# B&R Automation Studio project PT_KB_V01 (part 6)

#### ProcessValues.st
```iecst
ACTION ProcessValues:
	(* ======================================================================== *)
	(* 1) Izbor realnog protoka aktivnog izvora                                 *)
	(* ======================================================================== *)
	CASE PGRad.Ctrl.SelektovaniIzvor OF
		_01_BRB2:
			AktivniUlazniProtok := PG01_Remote.BRB2Sens.FtRB21.Value;

		_02_IEBKB1:
			AktivniUlazniProtok := IEB_KB1.Cntrl.Comm.Podstanica.Status.TrenutniProtok;

	ELSE
		AktivniUlazniProtok := 0.0;
	END_CASE

	(* ======================================================================== *)
	(* 2) Toplotne snage                                                        *)
	(* ======================================================================== *)
	Predata_Snaga := 4.181 * AktivniUlazniProtok
		* (PG.Sens.Tt._1.AI_Output.ScaledValue - PG.Sens.Tt._2.AI_Output.ScaledValue);
	Snaga_grejanja_hotela := 4.181 * AktivniUlazniProtok
		* (PG.Sens.Tt._1.AI_Output.ScaledValue - PG.Sens.Tt._4.AI_Output.ScaledValue);
	Snaga_sanitarnog_grejanja := Predata_Snaga - Snaga_grejanja_hotela;

	(* ======================================================================== *)
	(* 3) Ostale izvedene procesne velicine                                     *)
	(* ======================================================================== *)
	NivoPRihvatniSud := (PG.Sens.Pt._NS1.AI_Output.ScaledValue - PG.Sens.Pt._NS2.AI_Output.ScaledValue) / 0.09804;
	DP_strainer := PG.Sens.Pt._1.AI_Output.ScaledValue - PG.Sens.Pt._2.AI_Output.ScaledValue + 0.123;
	DP_Izmejnivac := PG.Sens.Pt._2.AI_Output.ScaledValue - PG.Sens.Pt._3.AI_Output.ScaledValue + 0.0015;
END_ACTION
```

### Program Logical/PID_Pu_01 (IEC)

#### Variables.var
```iecst
VAR
	Start_Pu_01 : BOOL;
END_VAR
```

#### Cyclic.st
```iecst
PROGRAM _CYCLIC
	(* ======================================================================== *)
	(* PID_Pu_01_CYCLIC                                                          *)
	(* Zatvorena petlja nivoa: ActValue uzima nivo prihvatnog suda,              *)
	(* a izlaz PID-a se, kada je dozvoljeno startPIDPu1, mapira na Pu._1 freq.   *)
	(* ======================================================================== *)

	(* -------------------------------------------------------------------------- *)
	(* 1) Rad po komandi state masine: PID je jedini vlasnik frekvencije i Run-a. *)
	(* -------------------------------------------------------------------------- *)
	IF PGRad_Cmd.Aktivan THEN
		Start_Pu_01 := FALSE;
		startPIDPu1 := PGRad_Cmd.PID.Enable;

		(* 1.1) Prenos procesnog zahteva u PID regulator. *)
		PID_Pu_01.Enable := PGRad_Cmd.PID.Enable;
		PID_Pu_01.ActValue := PGRad_Cmd.PID.ActValue;
		PID_Pu_01.SetValue := PGRad_Cmd.PID.SetValue;
		PID_Pu_01.Invert := PGRad_Cmd.PID.Invert;
		PID_Pu_01.MaxOut := PGRad_Cmd.PID.MaxOut;
		PID_Pu_01.EnableTracking := PGRad_Cmd.PID.EnableTracking;
		PID_Pu_01.TrackingValue := PGRad_Cmd.PID.TrackingValue;
		IF EDGEPOS(PGRad_Cmd.PID.Enable) THEN
			PID_Pu_01.Update := TRUE;
		END_IF
		PID_Pu_01();
		IF PID_Pu_01.UpdateDone THEN
			PID_Pu_01.Update := FALSE;
		END_IF

		(* 1.2) Iskljucivo izabrana izlazna pumpa dobija PID frekvenciju i Run. *)
		PG.Act.Pu._1.cmds.Run_fwd := FALSE;
		PG.Act.Pu._2.cmds.Run_fwd := FALSE;
		IF PGRad_Cmd.PID.Enable THEN
			IF PGRad_Cmd.Pumpe._01.Run THEN
				PG.Act.Pu._1.params.Freq := PID_Pu_01.Out;
				PG.Act.Pu._1.cmds.Run_fwd := TRUE;
			ELSIF PGRad_Cmd.Pumpe._02.Run THEN
				PG.Act.Pu._2.params.Freq := PID_Pu_01.Out;
				PG.Act.Pu._2.cmds.Run_fwd := TRUE;
			END_IF
		END_IF

	ELSE
		(* -------------------------------------------------------------------------- *)
		(* 2) Nasledjeni rucni/auto rad pumpe 1                                    *)
		(* -------------------------------------------------------------------------- *)
		(* 2.1) Ciklicni PID poziv sa nivoom prihvatnog suda kao merenom vrednoscu. *)
		PID_Pu_01.EnableTracking := FALSE;
		PID_Pu_01.ActValue := NivoPRihvatniSud;
		PID_Pu_01();

		IF startPIDPu1 THEN
			PG.Act.Pu._1.params.Freq := PID_Pu_01.Out;
		END_IF

		(* 2.2) Automatski start/stop iz nivoa i rucne komande. *)
		IF Pu_01_Auto THEN
			IF NivoPRihvatniSud > PID_Pu_01.SetValue THEN
				Start_Pu_01 := TRUE;
				startPIDPu1 := TRUE;
				PG.Act.AV._3.Open := TRUE;
			ELSIF (NivoPRihvatniSud < (PID_Pu_01.SetValue - 0.6))
				OR (NivoPRihvatniSud < 0.75) THEN
				Start_Pu_01 := FALSE;
				startPIDPu1 := FALSE;
				PG.Act.AV._3.Open := FALSE;
			END_IF
		END_IF

		IF EDGENEG(Pu_01_Auto) THEN
			Start_Pu_01 := FALSE;
		END_IF

		IF EDGEPOS(Start_Pu_01) THEN
			PID_Pu_01.Update := TRUE;
		END_IF

		(* 2.3) Primena Run komande i reset PID dozvole na ivicama zahteva. *)
		IF Start_Pu_01 THEN
			PID_Pu_01.Enable := TRUE;
			PG.Act.Pu._1.cmds.Run_fwd := TRUE;

			IF PID_Pu_01.UpdateDone THEN
				PID_Pu_01.Update := FALSE;
			END_IF
		END_IF

		IF EDGENEG(Start_Pu_01) THEN
			PID_Pu_01.Enable := FALSE;
			PG.Act.Pu._1.cmds.Run_fwd := FALSE;
		END_IF

		(* -------------------------------------------------------------------------- *)
		(* 3) Zadrzavanje otvorenog izlaznog ventila                                *)
		(* -------------------------------------------------------------------------- *)
		(* PG_V05 prati otvoren ulazni ventil PG_V01 u nasledjenom lokalnom rezimu. *)
		IF PG.Act.AV._1.Open THEN
			PG.Act.AV._5.Open := TRUE;
		END_IF
	END_IF
END_PROGRAM
```

#### Exit.st
```iecst
PROGRAM _EXIT
	(* ======================================================================== *)
	(* PID_Pu_01_EXIT                                                            *)
	(* Nema posebne EXIT akcije; Run i frekvencu vlasnicki postavlja CYCLIC.     *)
	(* ======================================================================== *)

END_PROGRAM
```

#### Init.st
```iecst
PROGRAM _INIT
	(* ======================================================================== *)
	(* PID_Pu_01_INIT                                                            *)
	(* U ovom tasku trenutno nema inicijalizacionih dodela.                      *)
	(* Retain procesni parametri se postavljaju iz HMI/visih nivoa logike.       *)
	(* ======================================================================== *)
	(* -------------------------------------------------------------------------- *)
	(* 1) Inicijalni parametri PID izlazne pumpe                                  *)
	(* -------------------------------------------------------------------------- *)
	(* Frekvencija izlazne pumpe je ogranicena na radni opseg 20.0..70.0 Hz. *)
	PID_Pu_01.MaxOut := 70.0; (* Gornja granica PID izlaza [Hz]. *)
	PID_Pu_01.MinOut := 20.0; (* Donja granica PID izlaza [Hz]. *)

	(* Parametri nivo regulacije; D deo je iskljucen, a filter prigusuje merenje. *)
	PID_Pu_01.PIDParameters.DerivativeTime := 0.0; (* D vreme [s]. *)
	PID_Pu_01.PIDParameters.FilterTime := 45.0; (* Filter merenja [s]. *)
	PID_Pu_01.PIDParameters.Gain := 96.3; (* Proporcionalno pojacanje. *)
	PID_Pu_01.PIDParameters.IntegrationTime := 180; (* Integraciono vreme [s]. *)
	PID_Pu_01.Invert := TRUE; (* Nivo regulacija koristi inverzni smer. *)

	PID_Pu_01.SetValue := 1.5; (* Lokalni pocetni setpoint nivoa [m]. *)

END_PROGRAM
```

### Program Logical/Rad_PG_KB (IEC)

#### Variables.var
```iecst
VAR
	(* Izvrsni kontekst state masine. *)
	State : E_PGRad_State := PG_00_Stand_By; (* Trenutni korak state masine *)
	Substep : USINT := 0; (* Podkorak aktivnog stanja: 0 = ulazak, 1..N = izvrsavanje *)

	(* HMI komande. *)
	KomandaStart : BOOL; (* HMI komanda za pokretanje sistema *)
	KomandaStop : BOOL; (* HMI komanda za kontrolisano zaustavljanje *)
	KomandaReset : BOOL; (* HMI komanda za reset uklonjene greske *)
	SelectIEBKB1 : BOOL; (* HMI Toggle: FALSE = BRB2, TRUE = IEBKB1; prihvata se samo u Standby. *)
	ManualMode : BOOL; (* Servisni rucni rezim; dozvoljen samo iz Standby. *)
	ManualSequence : USINT; (* Izabrana sekvenca servisnog rada. *)
	ManualStart : BOOL; (* Impuls za pokretanje izabrane sekvence. *)
	ManualStop : BOOL; (* Impuls za kontrolisani prekid servisne sekvence. *)
	ManualNextStep : BOOL; (* Impuls za sledeci dozvoljeni podkorak. *)
	ManualAbort : BOOL; (* Impuls za povratak u Standby. *)
	CmdSetDefaultParameters : BOOL; (* Jednokratno vracanje svih parametara na projektne default vrednosti *)

	(* Dijagnostika aktivne greske. *)
	FaultLatched : BOOL; (* Aktivna zakacena greska, zahteva reset nakon otklanjanja uzroka *)
	FaultCode : USINT; (* Sifra aktivne greske za HMI i AsIMA *)
	FaultText : STRING[80]; (* Tekst aktivne greske za HMI *)

	(* Nadzor polozaja ventila i protoka izvora. *)
	T_PG_V01_Close : TON; (* Timeout zatvaranja IEBKB1 dovodnog ventila. *)
	T_PG_V01_Open : TON; (* Timeout otvaranja IEBKB1 dovodnog ventila. *)
	T_PG_V02_Open : TON; (* Timeout otvaranja BRB2 dovodnog ventila pri pripremi BRB2. *)
	T_PG_V02_Close : TON; (* Timeout zatvaranja BRB2 dovodnog ventila pri pripremi IEBKB1. *)
	T_IEBKB1_StartProtokTimeout : TON; (* Maksimalno cekanje pocetka IEBKB1 dotoka nakon otvaranja PG_V05. *)
	T_IEBKB1_ProtokNula : TON; (* Debounce potvrda protoka manjeg od 0.1 l/s. *)
	T_IEBKB1_StopProtokTimeout : TON; (* Maksimalno cekanje prestanka IEBKB1 dotoka pre zatvaranja PG_V05. *)
	T_PG_V05_Close : TON; (* Timeout zatvaranja PG_V05 nakon potvrdenog prestanka IEBKB1 dotoka. *)

	(* PID regulatori i izvrsne pomocne vrednosti. *)
	T_PrelazPV05Cuvar : TON; (* Vreme mekane promene PT06 SP-a od preispiranja do cuvara instalacije. *)
	PID_PV05 : MTBasicsPID; (* PID PG_PV05: PT06 pritisak preispiranja i cuvara instalacije. *)
	PID_PV_UlazTanka : MTBasicsPID; (* PID aktivnog PG_PV01/PG_PV02: PT04 pritisak pri punjenju tanka. *)
	SP_PV05 : REAL; (* Trenutni rampirani PT06 SP za PID PG_PV05 [bar]. *)
	PV05IspiranjeOtvoreno : BOOL; (* PT06 je dostigao SP i PG_PV05 je dozvoljen za ispiranje. *)
	IzlaznaPumpaUStopu : BOOL; (* Pumpa nastavlja praznjenje tanka do donje granice hysteresis. *)
END_VAR
```

#### Cyclic.sfc
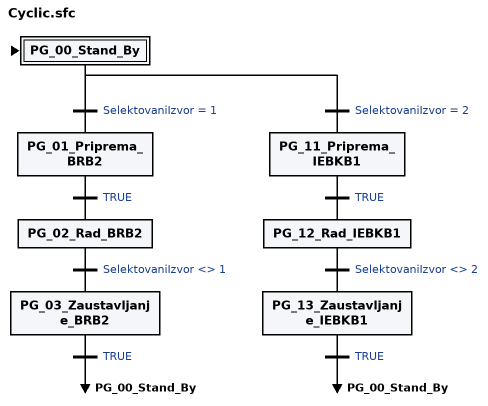
```iecst
PROGRAM _CYCLIC
INITIAL_STEP PG_00_Stand_By:
END_STEP
TRANSITION FROM PG_00_Stand_By TO PG_01_Priprema_BRB2:=
SelektovaniIzvor = 1
END_TRANSITION
TRANSITION FROM PG_00_Stand_By TO PG_11_Priprema_IEBKB1:=
SelektovaniIzvor = 2
END_TRANSITION
STEP PG_11_Priprema_IEBKB1:
END_STEP
TRANSITION FROM PG_11_Priprema_IEBKB1 TO PG_12_Rad_IEBKB1:=
TRUE
END_TRANSITION
STEP PG_12_Rad_IEBKB1:
END_STEP
TRANSITION FROM PG_12_Rad_IEBKB1 TO PG_13_Zaustavljanje_IEBKB1:=
SelektovaniIzvor <> 2
END_TRANSITION
STEP PG_13_Zaustavljanje_IEBKB1:
END_STEP
TRANSITION FROM PG_13_Zaustavljanje_IEBKB1 TO PG_00_Stand_By:=
TRUE
END_TRANSITION
(* @SFCISJUMP := 'PG_00_Stand_By' *)
STEP PG_01_Priprema_BRB2:
END_STEP
TRANSITION FROM PG_01_Priprema_BRB2 TO PG_02_Rad_BRB2:=
TRUE
END_TRANSITION
STEP PG_02_Rad_BRB2:
END_STEP
TRANSITION FROM PG_02_Rad_BRB2 TO PG_03_Zaustavljanje_BRB2:=
SelektovaniIzvor <> 1
END_TRANSITION
STEP PG_03_Zaustavljanje_BRB2:
END_STEP
TRANSITION FROM PG_03_Zaustavljanje_BRB2 TO PG_00_Stand_By:=
TRUE
END_TRANSITION
(* @SFCISJUMP := 'PG_00_Stand_By' *)
END_PROGRAM
```

#### Cyclic.st
```iecst
PROGRAM _CYCLIC
	(* ======================================================================== *)
	(* Rad_PG_KB_CYCLIC                                                          *)
	(* State masina izbora i rada izvora termalne vode: BRB2 (1) ili IEBKB1 (2). *)
	(* Prelazak izmedju grana ide iskljucivo preko PG_00_Stand_By - direktan     *)
	(* prelazak 1->2 ili 2->1 nije moguc.                                       *)
	(* ======================================================================== *)

	(* -------------------------------------------------------------------------- *)
	(* 1) Vracanje projektnih podrazumevanih parametara                          *)
	(* -------------------------------------------------------------------------- *)
	IF CmdSetDefaultParameters THEN
		PGRad.Par.SetPritisakPotisa := 1.5;
		PGRad.Par.MinProtok := 2.0;
		PGRad.Par.MaxProtok := 16.2;
		PGRad.Par.MinFR_Pumpe := 2.0;
		PGRad.Par.MaxFR_Pumpe := 16.2;
		PGRad.Par.SetPointNivoTanka := 1.5;
		PGRad.Par.SetPointMinTempIspiranja := 60.0;
		PGRad.Par.SetPointPritisakPV05Ispiranje := 5.5;
		PGRad.Par.SetPointPritisakUlazTanka := 5.5;
		PGRad.Par.SetPointMaxPritisakDolaznaCev := 6.5;
		PGRad.Par.TimeSP.PrelazPV05Cuvar_s := 15.0;
		PGRad.Par.PocetnaFrekvencaIzlaznePumpe := 20.0;
		PGRad.Par.MaxOtvorPropZaZatvaranje := 0.1;
		PGRad.Par.TimeSP.OverlapPumpi_s := 10.0;
		PGRad.Par.TimeSP.AutoRestartDelay_s := 60.0;
		PGRad.Par.TimeSP.ValvePositionTimeout_s := 30.0;
		PGRad.Par.TimeSP.InterlockDebounce_s := 2.0;

		(* BRB2 odzracivanje: oba ventila, prag 1.5 bar sa 0.5 bar histerezom. *)
		PGRad.Par.AirRelease.BRB2.PV03.NumberOfLS := 2;
		PGRad.Par.AirRelease.BRB2.PV03.PressureSP_bar := 1.5;
		PGRad.Par.AirRelease.BRB2.PV03.PressureHysteresis_bar := 0.5;
		PGRad.Par.AirRelease.BRB2.PV03.LS1.SP_Percent := 20.0;
		PGRad.Par.AirRelease.BRB2.PV03.LS1.Ramp_PercentPerSecond := 2.0;
		PGRad.Par.AirRelease.BRB2.PV03.LS1.ConfirmTime_s := 1.0;
		PGRad.Par.AirRelease.BRB2.PV03.LS2.SP_Percent := 89.0;
		PGRad.Par.AirRelease.BRB2.PV03.LS2.Ramp_PercentPerSecond := 15.0;
		PGRad.Par.AirRelease.BRB2.PV03.LS2.ConfirmTime_s := 1.0;
		PGRad.Par.AirRelease.BRB2.PV04 := PGRad.Par.AirRelease.BRB2.PV03;

		(* IEBKB1 odzracivanje: aktivan je PV03 sa nizim pragom pritiska. *)
		PGRad.Par.AirRelease.IEBKB1.PV03.NumberOfLS := 2;
		PGRad.Par.AirRelease.IEBKB1.PV03.PressureSP_bar := 0.15;
		PGRad.Par.AirRelease.IEBKB1.PV03.PressureHysteresis_bar := 0.05;
		PGRad.Par.AirRelease.IEBKB1.PV03.LS1.SP_Percent := 20.0;
		PGRad.Par.AirRelease.IEBKB1.PV03.LS1.Ramp_PercentPerSecond := 2.0;
		PGRad.Par.AirRelease.IEBKB1.PV03.LS1.ConfirmTime_s := 1.0;
		PGRad.Par.AirRelease.IEBKB1.PV03.LS2.SP_Percent := 89.0;
		PGRad.Par.AirRelease.IEBKB1.PV03.LS2.Ramp_PercentPerSecond := 15.0;
		PGRad.Par.AirRelease.IEBKB1.PV03.LS2.ConfirmTime_s := 1.0;
		PGRad.Par.AirRelease.IEBKB1.PV04 := PGRad.Par.AirRelease.IEBKB1.PV03;

		CmdSetDefaultParameters := FALSE;
	END_IF

	(* -------------------------------------------------------------------------- *)
	(* 2) Podrazumevane neretentivne komande po scan-u                            *)
	(* -------------------------------------------------------------------------- *)
	PGRad_Cmd.Aktivan := FALSE;
	PGRad_Cmd.Ventili._03_Open := FALSE;
	PGRad_Cmd.Ventili._04_Open := FALSE;
	PGRad_Cmd.Ventili._05_Open := FALSE;
	PGRad_Cmd.Ventili._06_Open := FALSE;
	PGRad_Cmd.Ventili._07_Open := FALSE;

	PGRad_Cmd.PropVentili.PV01.Enable := FALSE;
	PGRad_Cmd.PropVentili.PV01.SP_Percent := 0.0;
	PGRad_Cmd.PropVentili.PV02.Enable := FALSE;
	PGRad_Cmd.PropVentili.PV02.SP_Percent := 0.0;
	PGRad_Cmd.PropVentili.PV05.Enable := FALSE;
	PGRad_Cmd.PropVentili.PV05.SP_Percent := 0.0;
	PGRad_Cmd.AirRelease.PV03.Enable := FALSE;
	PGRad_Cmd.AirRelease.PV04.Enable := FALSE;
	PGRad_Cmd.AirRelease.UseIEBKB1Parameters := FALSE;
	PGRad_Cmd.AirRelease.ResetAll := KomandaReset;

	PGRad_Cmd.Pumpe._01.Run := FALSE;
	PGRad_Cmd.Pumpe._02.Run := FALSE;
	PGRad_Cmd.PID.Enable := FALSE;
	PGRad_Cmd.PID.ActValue := 0.0;
	PGRad_Cmd.PID.SetValue := 0.0;
	PGRad_Cmd.PID.Invert := FALSE;
	PGRad_Cmd.PID.MaxOut := 0.0;
	PGRad_Cmd.PID.EnableTracking := FALSE;
	PGRad_Cmd.PID.TrackingValue := 0.0;
	PGRad_BRB2Cmd.RadKaPodstanici := FALSE;
	PGRad_BRB2Cmd.ZahtevStarta := FALSE;
	PGRad_BRB2Cmd.ZahtevZaustavljanja := FALSE;
	PGRad_BRB2Cmd.ManualMode := ManualMode;
	PGRad_BRB2Cmd.ManualSequence := ManualSequence;
	PGRad_BRB2Cmd.ManualStart := ManualStart;
	PGRad_BRB2Cmd.ManualStop := ManualStop;
	PGRad_BRB2Cmd.ManualNextStep := ManualNextStep;
	PGRad_BRB2Cmd.ManualAbort := ManualAbort;
	PGRad_BRB2Cmd.VentiliPodstaniceZatvoreni := FALSE;
	PGRad_BRB2Cmd.PritisakIEBKB1 := IEB_KB1.Sens.Pt.B_02._01_value;
	PGRad_BRB2Cmd.PodstanicaURezimuRada := FALSE;
	IEB_KB1.Cntrl.Comm.Podstanica.Zahtev.ZahtevVode := FALSE;
	IEB_KB1.Cntrl.Comm.Podstanica.Zahtev.NivoPrihvatnogTanka := NivoPRihvatniSud;
	IEB_KB1.Cntrl.Comm.Podstanica.Zahtev.CiljaniProtok := PGRad.Par.MaxProtok;
	IEB_KB1.Cntrl.Comm.Podstanica.Zahtev.ModRada := 0;
	IEB_KB1.Cntrl.proba := FALSE;

	(* Izbor izvora sa HMI prihvata se samo u bezbednom Standby stanju. *)
	IF State = PG_00_Stand_By THEN
		IF SelectIEBKB1 THEN
			PGRad.Ctrl.SelektovaniIzvor := _02_IEBKB1;
		ELSE
			PGRad.Ctrl.SelektovaniIzvor := _01_BRB2;
		END_IF;
	ELSE
		SelectIEBKB1 := PGRad.Ctrl.SelektovaniIzvor = _02_IEBKB1;
	END_IF;

	(* -------------------------------------------------------------------------- *)
	(* 3) Tajmeri pripreme BRB2 dovodne putanje                                  *)
	(* -------------------------------------------------------------------------- *)
	T_PG_V01_Close.IN := FALSE;
	T_PG_V01_Close.PT := REAL_TO_TIME(PGRad.Par.TimeSP.ValvePositionTimeout_s * 1000.0);
	T_PG_V02_Open.IN := FALSE;
	T_PG_V02_Open.PT := REAL_TO_TIME(PGRad.Par.TimeSP.ValvePositionTimeout_s * 1000.0);
	T_PG_V02_Close.IN := FALSE;
	T_PG_V02_Close.PT := REAL_TO_TIME(PGRad.Par.TimeSP.ValvePositionTimeout_s * 1000.0);
	T_PG_V01_Open.IN := FALSE;
	T_PG_V01_Open.PT := REAL_TO_TIME(PGRad.Par.TimeSP.ValvePositionTimeout_s * 1000.0);
	T_IEBKB1_StartProtokTimeout.IN := FALSE;
	T_IEBKB1_StartProtokTimeout.PT := REAL_TO_TIME(PGRad.Par.TimeSP.ValvePositionTimeout_s * 1000.0);
	T_IEBKB1_ProtokNula.IN := FALSE;
	T_IEBKB1_ProtokNula.PT := REAL_TO_TIME(PGRad.Par.TimeSP.InterlockDebounce_s * 1000.0);
	T_IEBKB1_StopProtokTimeout.IN := FALSE;
	T_IEBKB1_StopProtokTimeout.PT := REAL_TO_TIME(PGRad.Par.TimeSP.ValvePositionTimeout_s * 1000.0);
	T_PG_V05_Close.IN := FALSE;
	T_PG_V05_Close.PT := REAL_TO_TIME(PGRad.Par.TimeSP.ValvePositionTimeout_s * 1000.0);
	T_PrelazPV05Cuvar.IN := FALSE;
	T_PrelazPV05Cuvar.PT := REAL_TO_TIME(PGRad.Par.TimeSP.PrelazPV05Cuvar_s * 1000.0);

	CASE State OF

		PG_00_Stand_By:
			(* Neretentivni vektor je bezbedno resetovan u sekciji 2; V01/V02 se ne menjaju. *)
			PV05IspiranjeOtvoreno := FALSE;
			(* Start je dozvoljen samo sa izabranim izvorom i regulacionom varijantom. *)
			IF ManualMode AND ManualStart AND (ManualSequence = 1) THEN
				PGRad.Ctrl.SelektovaniIzvor := _01_BRB2;
				ManualStart := FALSE;
				State := PG_01_Priprema_BRB2;
				Substep := 0;
			ELSIF ManualMode AND ManualStart AND (ManualSequence = 2) THEN
				PGRad.Ctrl.SelektovaniIzvor := _02_IEBKB1;
				ManualStart := FALSE;
				State := PG_11_Priprema_IEBKB1;
				Substep := 0;
			ELSIF KomandaStart
				AND (NOT ManualMode)
				AND (NOT FaultLatched)
				AND (PGRad.Ctrl.RegulacionaVarijanta <> _00_neaktivan)
				AND (PGRad.Ctrl.SelektovaniIzvor = _01_BRB2) THEN
				State := PG_01_Priprema_BRB2;
				Substep := 0;
			ELSIF KomandaStart
				AND (NOT FaultLatched)
				AND (PGRad.Ctrl.RegulacionaVarijanta <> _00_neaktivan)
				AND (PGRad.Ctrl.SelektovaniIzvor = _02_IEBKB1) THEN
				State := PG_11_Priprema_IEBKB1;
				Substep := 0;
			END_IF

		PG_01_Priprema_BRB2:
			IF ManualStop OR ManualAbort THEN
				KomandaStop := TRUE;
				ManualStop := FALSE;
				ManualAbort := FALSE;
			END_IF;
			PGRad_BRB2Cmd.RadKaPodstanici := TRUE;
			PGRad_BRB2Cmd.ZahtevStarta := TRUE;
			CASE Substep OF
				0:
					(* Prioritet BRB2: najpre zatvori dovod sa IEBKB1. *)
					PGRad.CmdRetain.V01_Open := FALSE;
					Substep := 1;

				1:
					(* Otvaranje BRB2 dovoda je dozvoljeno tek po potvrdi zatvorenog V01. *)
					PGRad.CmdRetain.V01_Open := FALSE;
					T_PG_V01_Close.IN := NOT PG.Act.AV._1.Closed;
					IF PG.Act.AV._1.Closed AND (NOT ManualMode OR ManualNextStep) THEN
						ManualNextStep := FALSE;
						PGRad.CmdRetain.V02_Open := TRUE;
						Substep := 2;
					ELSIF T_PG_V01_Close.Q THEN
						PGRad.CmdRetain.V01_Open := FALSE;
						PGRad.CmdRetain.V02_Open := FALSE;
						FaultLatched := TRUE;
						FaultCode := 11;
						FaultText := 'PG_V01 nije zatvoren za zadato vreme';
						State := PG_00_Stand_By;
						Substep := 0;
					END_IF

				2:
					(* Ceka se fizicka potvrda otvorenog BRB2 dovoda. *)
					PGRad.CmdRetain.V01_Open := FALSE;
					PGRad.CmdRetain.V02_Open := TRUE;
					T_PG_V02_Open.IN := NOT PG.Act.AV._2.Opened;
					IF PG.Act.AV._2.Opened AND (NOT ManualMode OR ManualNextStep) THEN
						ManualNextStep := FALSE;
						Substep := 3;
					ELSIF T_PG_V02_Open.Q THEN
						PGRad.CmdRetain.V01_Open := FALSE;
						PGRad.CmdRetain.V02_Open := FALSE;
						FaultLatched := TRUE;
						FaultCode := 12;
						FaultText := 'PG_V02 nije otvoren za zadato vreme';
						State := PG_00_Stand_By;
						Substep := 0;
					END_IF

				3:
					(* PG_PV05 se otvara nakon dostignutog PT06 pritiska; temperatura se proverava tek posle BRB2 minimuma. *)
					IF PG.Sens.Pt._6.AI_Output.ScaledValue >= PGRad.Par.SetPointPritisakPV05Ispiranje THEN
						PV05IspiranjeOtvoreno := TRUE;
					END_IF;
					IF PV05IspiranjeOtvoreno THEN
						PGRad_Cmd.Aktivan := TRUE;
						PGRad_Cmd.PropVentili.PV05.Enable := TRUE;
					END_IF;
					IF PGRad_BRB2.IspiranjeMinTrajanjeDostignuto
						AND (PG.Sens.Tt._7.AI_Output.ScaledValue >= PGRad.Par.SetPointMinTempIspiranja) THEN
						IF ManualMode AND NOT ManualNextStep THEN
							(* Manual mode holds the completed rinse step until operator confirmation. *)
						ELSE
							ManualNextStep := FALSE;
							IF ManualMode AND (ManualSequence = 1) THEN
								(* Manual flush ends here; controlled stop closes the BRB2 path. *)
								KomandaStop := TRUE;
								State := PG_03_Zaustavljanje_BRB2;
								Substep := 0;
							ELSE
								Substep := 4;
							END_IF
						END_IF
					END_IF

				4:
					(* Priprema puta ka tanku: otvara se samo ON/OFF ventil izabranog ulaznog PV-a. *)
					PGRad_Cmd.Aktivan := TRUE;
					PGRad_Cmd.PropVentili.PV05.Enable := TRUE;
					CASE PGRad.Ctrl.AktivniPropVentilUlazTanka OF
						_01_PG_PV01:
							PGRad_Cmd.Ventili._06_Open := TRUE;
							PGRad_Cmd.PropVentili.PV01.Enable := TRUE;
							Substep := 5;
						_02_PG_PV02:
							PGRad_Cmd.Ventili._07_Open := TRUE;
							PGRad_Cmd.PropVentili.PV02.Enable := TRUE;
							Substep := 5;
					END_CASE

				5:
					(* Mek prelaz: ulazni PV vodi PT04, a PT06 SP PG_PV05 raste 5.5 -> 6.5 bar. *)
					PGRad_Cmd.Aktivan := TRUE;
					PGRad_Cmd.PropVentili.PV05.Enable := TRUE;
					T_PrelazPV05Cuvar.IN := TRUE;
					CASE PGRad.Ctrl.AktivniPropVentilUlazTanka OF
						_01_PG_PV01:
							PGRad_Cmd.Ventili._06_Open := TRUE;
							PGRad_Cmd.PropVentili.PV01.Enable := TRUE;
						_02_PG_PV02:
							PGRad_Cmd.Ventili._07_Open := TRUE;
							PGRad_Cmd.PropVentili.PV02.Enable := TRUE;
					END_CASE
					IF T_PrelazPV05Cuvar.Q AND (NOT ManualMode OR ManualNextStep) THEN
						ManualNextStep := FALSE;
						Substep := 6;
					END_IF

				6:
					(* Punjenje tanka: PV05 je cuvar PT06, a aktivni ulazni PV odrzava PT04. *)
					PGRad_Cmd.Aktivan := TRUE;
					PGRad_Cmd.PropVentili.PV05.Enable := TRUE;
					CASE PGRad.Ctrl.AktivniPropVentilUlazTanka OF
						_01_PG_PV01:
							PGRad_Cmd.Ventili._06_Open := TRUE;
							PGRad_Cmd.PropVentili.PV01.Enable := TRUE;
						_02_PG_PV02:
							PGRad_Cmd.Ventili._07_Open := TRUE;
							PGRad_Cmd.PropVentili.PV02.Enable := TRUE;
					END_CASE
					IF (NivoPRihvatniSud >= PGRad.Par.SetPointNivoTanka)
						AND (NOT ManualMode OR ManualNextStep) THEN
						ManualNextStep := FALSE;
						State := PG_02_Rad_BRB2;
						Substep := 0;
					END_IF

			ELSE
				Substep := 0;
			END_CASE

		PG_02_Rad_BRB2:
			PGRad_BRB2Cmd.RadKaPodstanici := TRUE;
			PGRad_BRB2Cmd.ZahtevStarta := TRUE;
			(* Odrzava PID regulaciju ulaza i PT06 cuvara nakon punjenja tanka. *)
			PGRad_Cmd.Aktivan := TRUE;
			PGRad_Cmd.PropVentili.PV05.Enable := TRUE;
			CASE PGRad.Ctrl.AktivniPropVentilUlazTanka OF
				_01_PG_PV01:
					PGRad_Cmd.Ventili._06_Open := TRUE;
					PGRad_Cmd.PropVentili.PV01.Enable := TRUE;
				_02_PG_PV02:
					PGRad_Cmd.Ventili._07_Open := TRUE;
					PGRad_Cmd.PropVentili.PV02.Enable := TRUE;
			END_CASE

			(* Izlaznu pumpu pokrece i frekvencu vodi iskljucivo PID_Pu_01. *)
			CASE PGRad.Ctrl.RegulacionaVarijanta OF
				_01_REG_PRITISAK:
					PGRad_Cmd.PID.Enable := TRUE;
					PGRad_Cmd.PID.ActValue := PG.Sens.Pt._5.AI_Output.ScaledValue;
					PGRad_Cmd.PID.SetValue := PGRad.Par.SetPritisakPotisa;
					PGRad_Cmd.PID.Invert := FALSE;
				_02_REG_NIVO:
					PGRad_Cmd.PID.Enable := TRUE;
					PGRad_Cmd.PID.ActValue := NivoPRihvatniSud;
					PGRad_Cmd.PID.SetValue := PGRad.Par.SetPointNivoTanka;
					PGRad_Cmd.PID.Invert := TRUE;
			END_CASE

			IF PGRad_Cmd.PID.Enable THEN
				PGRad_Cmd.PID.TrackingValue := PGRad.Par.PocetnaFrekvencaIzlaznePumpe;
				PGRad_Cmd.PID.EnableTracking := (Substep = 0);
				CASE PGRad.Ctrl.AktivnaPumpaIzlazTanka OF
					_01_Pu_PG_01:
						PGRad_Cmd.Ventili._03_Open := TRUE;
						PGRad_Cmd.Pumpe._01.Run := TRUE;
						PGRad_Cmd.PID.MaxOut := 70.0;
					_02_Pu_PG_02:
						PGRad_Cmd.Ventili._04_Open := TRUE;
						PGRad_Cmd.Pumpe._02.Run := TRUE;
						PGRad_Cmd.PID.MaxOut := 50.0;
				END_CASE
				Substep := 1;
			END_IF

			(* BRB2 sme preci u rad tek kada je tank pun i izabrana PG pumpa stvarno radi. *)
			PGRad_BRB2Cmd.PodstanicaURezimuRada :=
				(NivoPRihvatniSud >= PGRad.Par.SetPointNivoTanka)
				AND (
					((PGRad.Ctrl.AktivnaPumpaIzlazTanka = _01_Pu_PG_01)
						AND PG.Act.Pu._1.states.RUN)
					OR ((PGRad.Ctrl.AktivnaPumpaIzlazTanka = _02_Pu_PG_02)
						AND PG.Act.Pu._2.states.RUN)
				);

			(* Napusta granu cim PGRad.Ctrl.SelektovaniIzvor vise nije _01_BRB2. *)
			IF KomandaStop OR (PGRad.Ctrl.SelektovaniIzvor <> _01_BRB2) THEN
				State := PG_03_Zaustavljanje_BRB2;
				Substep := 0;
			END_IF

		PG_03_Zaustavljanje_BRB2:
			(* PT najpre trazi BRB2 ramp-down, zatim zatvara PV grane po stop SP potvrdi. *)
			PGRad_Cmd.Aktivan := TRUE;
			PGRad_BRB2Cmd.ZahtevZaustavljanja := TRUE;

			IF Substep = 0 THEN
				IzlaznaPumpaUStopu := TRUE;
				Substep := 1;
			END_IF;

			(* Izlazna pumpa ostaje na aktivnoj regulaciji dok tank ne padne ispod 60% SP-a. *)
			IF NivoPRihvatniSud < (0.6 * PGRad.Par.SetPointNivoTanka) THEN
				IzlaznaPumpaUStopu := FALSE;
			END_IF;

			IF IzlaznaPumpaUStopu THEN
				CASE PGRad.Ctrl.RegulacionaVarijanta OF
					_01_REG_PRITISAK:
						PGRad_Cmd.PID.Enable := TRUE;
						PGRad_Cmd.PID.ActValue := PG.Sens.Pt._5.AI_Output.ScaledValue;
						PGRad_Cmd.PID.SetValue := PGRad.Par.SetPritisakPotisa;
						PGRad_Cmd.PID.Invert := FALSE;
					_02_REG_NIVO:
						PGRad_Cmd.PID.Enable := TRUE;
						PGRad_Cmd.PID.ActValue := NivoPRihvatniSud;
						PGRad_Cmd.PID.SetValue := PGRad.Par.SetPointNivoTanka;
						PGRad_Cmd.PID.Invert := TRUE;
				END_CASE

				CASE PGRad.Ctrl.AktivnaPumpaIzlazTanka OF
					_01_Pu_PG_01:
						PGRad_Cmd.Ventili._03_Open := TRUE;
						PGRad_Cmd.Pumpe._01.Run := TRUE;
						PGRad_Cmd.PID.MaxOut := 70.0;
					_02_Pu_PG_02:
						PGRad_Cmd.Ventili._04_Open := TRUE;
						PGRad_Cmd.Pumpe._02.Run := TRUE;
						PGRad_Cmd.PID.MaxOut := 50.0;
				END_CASE
			END_IF;

			IF NOT PGRad_BRB2.StopSPDostignut THEN
				(* Dok BRB2 spusta frekvenciju, PT06 i PT04 ostaju u regulaciji. *)
				PGRad_Cmd.PropVentili.PV05.Enable := TRUE;
				CASE PGRad.Ctrl.AktivniPropVentilUlazTanka OF
					_01_PG_PV01:
						PGRad_Cmd.Ventili._06_Open := TRUE;
						PGRad_Cmd.PropVentili.PV01.Enable := TRUE;
					_02_PG_PV02:
						PGRad_Cmd.Ventili._07_Open := TRUE;
						PGRad_Cmd.PropVentili.PV02.Enable := TRUE;
				END_CASE
			END_IF;

			(* Nakon BRB2 stop SP-a svi proporcionalni ventili ostaju bez zahteva. *)
			PGRad_BRB2Cmd.VentiliPodstaniceZatvoreni := PGRad_BRB2.StopSPDostignut
				AND (PG.Act.PV._1.PV_Output.PV_Percent <= PGRad.Par.MaxOtvorPropZaZatvaranje)
				AND (PG.Act.PV._2.PV_Output.PV_Percent <= PGRad.Par.MaxOtvorPropZaZatvaranje)
				AND (PG.Act.PV._5.PV_Output.PV_Percent <= PGRad.Par.MaxOtvorPropZaZatvaranje);

			IF PGRad_BRB2.RB2V02Zatvoren AND NOT IzlaznaPumpaUStopu THEN
				State := PG_00_Stand_By;
				Substep := 0;
			END_IF

		PG_11_Priprema_IEBKB1:
			(* IEBKB1 put koristi samo PG_V01 i PG_V05; PV01/PV02/V06/V07 ostaju zatvoreni. *)
			IEB_KB1.Cntrl.Comm.Podstanica.Zahtev.ZahtevVode := TRUE;
			IEB_KB1.Cntrl.Comm.Podstanica.Zahtev.ModRada := 1;
			IEB_KB1.Cntrl.proba := TRUE;
			CASE Substep OF
				0:
					PGRad.CmdRetain.V02_Open := FALSE;
					Substep := 1;

				1:
					PGRad.CmdRetain.V02_Open := FALSE;
					T_PG_V02_Close.IN := NOT PG.Act.AV._2.Closed;
					IF PG.Act.AV._2.Closed THEN
						PGRad.CmdRetain.V01_Open := TRUE;
						Substep := 2;
					ELSIF T_PG_V02_Close.Q THEN
						PGRad.CmdRetain.V01_Open := FALSE;
						PGRad.CmdRetain.V02_Open := FALSE;
						FaultLatched := TRUE;
						FaultCode := 13;
						FaultText := 'PG_V02 nije zatvoren za zadato vreme';
						State := PG_00_Stand_By;
						Substep := 0;
					END_IF

				2:
					PGRad.CmdRetain.V01_Open := TRUE;
					PGRad.CmdRetain.V02_Open := FALSE;
					T_PG_V01_Open.IN := NOT PG.Act.AV._1.Opened;
					IF PG.Act.AV._1.Opened THEN
						Substep := 3;
					ELSIF T_PG_V01_Open.Q THEN
						PGRad.CmdRetain.V01_Open := FALSE;
						FaultLatched := TRUE;
						FaultCode := 14;
						FaultText := 'PG_V01 nije otvoren za zadato vreme';
						State := PG_00_Stand_By;
						Substep := 0;
					END_IF

				3:
					(* V05 vodi IEBKB1 vodu direktno u prihvatni tank. *)
					PGRad_Cmd.Aktivan := TRUE;
					PGRad_Cmd.Ventili._05_Open := TRUE;
					T_IEBKB1_StartProtokTimeout.IN :=
						IEB_KB1.Cntrl.Comm.Podstanica.Status.TrenutniProtok <= 0.1;
					IF IEB_KB1.Cntrl.Comm.Podstanica.Status.TrenutniProtok > 0.1 THEN
						Substep := 4;
					ELSIF T_IEBKB1_StartProtokTimeout.Q THEN
						FaultLatched := TRUE;
						FaultCode := 18;
						FaultText := 'IEBKB1 dotok nije poceo za zadato vreme';
						State := PG_13_Zaustavljanje_IEBKB1;
						Substep := 0;
					END_IF

				4:
					PGRad_Cmd.Aktivan := TRUE;
					PGRad_Cmd.Ventili._05_Open := TRUE;
					IF NivoPRihvatniSud >= PGRad.Par.SetPointNivoTanka THEN
						State := PG_12_Rad_IEBKB1;
						Substep := 0;
					END_IF

			ELSE
				Substep := 0;
			END_CASE

		PG_12_Rad_IEBKB1:
			(* IEBKB1 dovod ostaje otvoren; PT lokalno vodi samo izlaznu pumpu. *)
			PGRad.CmdRetain.V01_Open := TRUE;
			PGRad.CmdRetain.V02_Open := FALSE;
			PGRad_Cmd.Aktivan := TRUE;
			PGRad_Cmd.Ventili._05_Open := TRUE;
			IEB_KB1.Cntrl.Comm.Podstanica.Zahtev.ZahtevVode := TRUE;
			IEB_KB1.Cntrl.Comm.Podstanica.Zahtev.ModRada := 2;
			IEB_KB1.Cntrl.proba := TRUE;

			CASE PGRad.Ctrl.RegulacionaVarijanta OF
				_01_REG_PRITISAK:
					PGRad_Cmd.PID.Enable := TRUE;
					PGRad_Cmd.PID.ActValue := PG.Sens.Pt._5.AI_Output.ScaledValue;
					PGRad_Cmd.PID.SetValue := PGRad.Par.SetPritisakPotisa;
					PGRad_Cmd.PID.Invert := FALSE;
				_02_REG_NIVO:
					PGRad_Cmd.PID.Enable := TRUE;
					PGRad_Cmd.PID.ActValue := NivoPRihvatniSud;
					PGRad_Cmd.PID.SetValue := PGRad.Par.SetPointNivoTanka;
					PGRad_Cmd.PID.Invert := TRUE;
			END_CASE

			IF PGRad_Cmd.PID.Enable THEN
				PGRad_Cmd.PID.TrackingValue := PGRad.Par.PocetnaFrekvencaIzlaznePumpe;
				PGRad_Cmd.PID.EnableTracking := (Substep = 0);
				CASE PGRad.Ctrl.AktivnaPumpaIzlazTanka OF
					_01_Pu_PG_01:
						PGRad_Cmd.Ventili._03_Open := TRUE;
						PGRad_Cmd.Pumpe._01.Run := TRUE;
						PGRad_Cmd.PID.MaxOut := 70.0;
					_02_Pu_PG_02:
						PGRad_Cmd.Ventili._04_Open := TRUE;
						PGRad_Cmd.Pumpe._02.Run := TRUE;
						PGRad_Cmd.PID.MaxOut := 50.0;
				END_CASE
				Substep := 1;
			END_IF

			IF KomandaStop OR (PGRad.Ctrl.SelektovaniIzvor <> _02_IEBKB1) THEN
				State := PG_13_Zaustavljanje_IEBKB1;
				Substep := 0;
			END_IF

		PG_13_Zaustavljanje_IEBKB1:
			(* ==================================================================== *)
			(* 1) Podrazumevane komande za kontrolisano zaustavljanje IEBKB1       *)
			(* ==================================================================== *)
			(* Zahtev bunaru je uklonjen; V05 ostaje otvoren do potvrdenog nultog protoka. *)
			PGRad_Cmd.Aktivan := TRUE;
			PGRad.CmdRetain.V02_Open := FALSE;
			IEB_KB1.Cntrl.Comm.Podstanica.Zahtev.ModRada := 3;
			IEB_KB1.Cntrl.proba := FALSE;

			(* ==================================================================== *)
			(* 2) Zadrzavanje rada izlazne pumpe dok se tank ne isprazni            *)
			(* ==================================================================== *)
			IF Substep = 0 THEN
				IzlaznaPumpaUStopu := TRUE;
				Substep := 1;
			END_IF;

			IF NivoPRihvatniSud < (0.6 * PGRad.Par.SetPointNivoTanka) THEN
				IzlaznaPumpaUStopu := FALSE;
			END_IF;

			IF IzlaznaPumpaUStopu THEN
				CASE PGRad.Ctrl.RegulacionaVarijanta OF
					_01_REG_PRITISAK:
						PGRad_Cmd.PID.Enable := TRUE;
						PGRad_Cmd.PID.ActValue := PG.Sens.Pt._5.AI_Output.ScaledValue;
						PGRad_Cmd.PID.SetValue := PGRad.Par.SetPritisakPotisa;
						PGRad_Cmd.PID.Invert := FALSE;
					_02_REG_NIVO:
						PGRad_Cmd.PID.Enable := TRUE;
						PGRad_Cmd.PID.ActValue := NivoPRihvatniSud;
						PGRad_Cmd.PID.SetValue := PGRad.Par.SetPointNivoTanka;
						PGRad_Cmd.PID.Invert := TRUE;
				END_CASE

				CASE PGRad.Ctrl.AktivnaPumpaIzlazTanka OF
					_01_Pu_PG_01:
						PGRad_Cmd.Ventili._03_Open := TRUE;
						PGRad_Cmd.Pumpe._01.Run := TRUE;
						PGRad_Cmd.PID.MaxOut := 70.0;
					_02_Pu_PG_02:
						PGRad_Cmd.Ventili._04_Open := TRUE;
						PGRad_Cmd.Pumpe._02.Run := TRUE;
						PGRad_Cmd.PID.MaxOut := 50.0;
				END_CASE
			END_IF

			(* ==================================================================== *)
			(* 3) Stop podkoraci: nulti protok, PG_V05, zatim PG_V01                *)
			(* ==================================================================== *)
			CASE Substep OF
				1:
					PGRad.CmdRetain.V01_Open := TRUE;
					PGRad_Cmd.Ventili._05_Open := TRUE;
					T_IEBKB1_ProtokNula.IN := IEB_KB1.Sens.MP.B_01._01_value < 0.1;
					T_IEBKB1_StopProtokTimeout.IN := NOT T_IEBKB1_ProtokNula.Q;
					IF T_IEBKB1_ProtokNula.Q THEN
						Substep := 2;
					ELSIF T_IEBKB1_StopProtokTimeout.Q THEN
						FaultLatched := TRUE;
						FaultCode := 16;
						FaultText := 'IEBKB1 dotok nije prestao za zadato vreme';
					END_IF

				2:
					(* PG_V05 se zatvara tek nakon stabilne potvrde nultog dotoka. *)
					T_PG_V05_Close.IN := NOT PG.Act.AV._5.Closed;
					IF PG.Act.AV._5.Closed THEN
						IF PGRad.Ctrl.SelektovaniIzvor = _02_IEBKB1 THEN
							IF NOT IzlaznaPumpaUStopu THEN
								State := PG_00_Stand_By;
								Substep := 0;
							END_IF
						ELSE
							PGRad.CmdRetain.V01_Open := FALSE;
							Substep := 3;
						END_IF
					ELSIF T_PG_V05_Close.Q THEN
						FaultLatched := TRUE;
						FaultCode := 17;
						FaultText := 'PG_V05 nije zatvoren za zadato vreme';
					END_IF

				3:
					(* V01 se zatvara samo kada je zadrzani izbor izvora promenjen. *)
					PGRad.CmdRetain.V01_Open := FALSE;
					T_PG_V01_Close.IN := NOT PG.Act.AV._1.Closed;
					IF PG.Act.AV._1.Closed AND NOT IzlaznaPumpaUStopu THEN
						State := PG_00_Stand_By;
						Substep := 0;
					ELSIF T_PG_V01_Close.Q THEN
						FaultLatched := TRUE;
						FaultCode := 15;
						FaultText := 'PG_V01 nije zatvoren za zadato vreme';
					END_IF

			ELSE
				Substep := 0;
			END_CASE

	ELSE
		(* Nepoznato stanje - bezbedan povratak na Stand_By. *)
		State := PG_00_Stand_By;

	END_CASE

	(* -------------------------------------------------------------------------- *)
	(* 4) Rezim rada i dozvole odzracivanja                                      *)
	(* -------------------------------------------------------------------------- *)
	(* Tokom pripreme, rada i zaustavljanja zadrzava se parametarski skup izvora. *)
	CASE State OF
		PG_01_Priprema_BRB2, PG_02_Rad_BRB2, PG_03_Zaustavljanje_BRB2:
			PGRad_Cmd.AirRelease.PV03.Enable := TRUE;
			PGRad_Cmd.AirRelease.PV04.Enable := TRUE;
			PGRad_Cmd.AirRelease.UseIEBKB1Parameters := FALSE;
		PG_11_Priprema_IEBKB1, PG_12_Rad_IEBKB1, PG_13_Zaustavljanje_IEBKB1:
			PGRad_Cmd.AirRelease.PV03.Enable := TRUE;
			PGRad_Cmd.AirRelease.PV04.Enable := FALSE;
			PGRad_Cmd.AirRelease.UseIEBKB1Parameters := TRUE;
	END_CASE

	(* -------------------------------------------------------------------------- *)
	(* 5) Izvrsavanje tajmera pripreme, stop sekvence i prelaza PV05              *)
	(* -------------------------------------------------------------------------- *)
	(* IN/PT su pripremljeni u sekciji 3 i aktivnom stanju; ovde se osvezava Q/ET. *)
	T_PG_V01_Close();
	T_PG_V01_Open();
	T_PG_V02_Open();
	T_PG_V02_Close();
	T_IEBKB1_StartProtokTimeout();
	T_IEBKB1_ProtokNula();
	T_IEBKB1_StopProtokTimeout();
	T_PG_V05_Close();
	T_PrelazPV05Cuvar();

	(* -------------------------------------------------------------------------- *)
	(* 6) PID petlje proporcionalnih ventila                                     *)
	(* -------------------------------------------------------------------------- *)
	(* 6.1) PV05 cuva PT06 tokom punjenja, rada BRB2 i njegovog ramp-down-a. *)
	PID_PV05.Enable := ((State = PG_01_Priprema_BRB2) AND (Substep >= 3))
		OR (State = PG_02_Rad_BRB2)
		OR ((State = PG_03_Zaustavljanje_BRB2) AND NOT PGRad_BRB2.StopSPDostignut);
	PID_PV05.ActValue := PG.Sens.Pt._6.AI_Output.ScaledValue; (* Merena vrednost PT06. *)
	(* U prelazu se SP linearno podize od ispiranja do maksimalnog pritiska voda. *)
	IF (State = PG_01_Priprema_BRB2) AND (Substep = 5) THEN
		SP_PV05 := PGRad.Par.SetPointPritisakPV05Ispiranje
			+ ((PGRad.Par.SetPointMaxPritisakDolaznaCev - PGRad.Par.SetPointPritisakPV05Ispiranje)
			* TIME_TO_REAL(T_PrelazPV05Cuvar.ET) / TIME_TO_REAL(T_PrelazPV05Cuvar.PT));
	ELSIF (((State = PG_01_Priprema_BRB2) AND (Substep >= 6))
		OR (State = PG_02_Rad_BRB2)
		OR ((State = PG_03_Zaustavljanje_BRB2) AND NOT PGRad_BRB2.StopSPDostignut)) THEN
		SP_PV05 := PGRad.Par.SetPointMaxPritisakDolaznaCev;
	ELSE
		SP_PV05 := PGRad.Par.SetPointPritisakPV05Ispiranje;
	END_IF
	PID_PV05.SetValue := SP_PV05; (* Izracunati SP pritiska dolaznog voda. *)
	PID_PV05();
	IF PID_PV05.UpdateDone THEN
		PID_PV05.Update := FALSE;
	END_IF

	(* 6.2) Aktivni ulazni ventil tanka odrzava PT04 po zadrzanom setpoint-u. *)
	PID_PV_UlazTanka.Enable := ((State = PG_01_Priprema_BRB2) AND (Substep >= 4))
		OR (State = PG_02_Rad_BRB2)
		OR ((State = PG_03_Zaustavljanje_BRB2) AND NOT PGRad_BRB2.StopSPDostignut);
	PID_PV_UlazTanka.ActValue := PG.Sens.Pt._4.AI_Output.ScaledValue; (* Merena vrednost PT04. *)
	PID_PV_UlazTanka.SetValue := PGRad.Par.SetPointPritisakUlazTanka; (* Zadrzani PT04 SP. *)
	PID_PV_UlazTanka();
	IF PID_PV_UlazTanka.UpdateDone THEN
		PID_PV_UlazTanka.Update := FALSE;
	END_IF

	(* 6.3) PID izlazi se upisuju samo kada odgovarajuca sekvenca dozvoljava ventil. *)
	IF (((State = PG_01_Priprema_BRB2) AND (Substep >= 3))
		OR (State = PG_02_Rad_BRB2)
		OR ((State = PG_03_Zaustavljanje_BRB2) AND NOT PGRad_BRB2.StopSPDostignut)) THEN
		PGRad_Cmd.PropVentili.PV05.SP_Percent := PID_PV05.Out;
	END_IF
	IF (((State = PG_01_Priprema_BRB2) AND (Substep >= 4))
		OR (State = PG_02_Rad_BRB2)
		OR ((State = PG_03_Zaustavljanje_BRB2) AND NOT PGRad_BRB2.StopSPDostignut)) THEN
		CASE PGRad.Ctrl.AktivniPropVentilUlazTanka OF
			_01_PG_PV01:
				PGRad_Cmd.PropVentili.PV01.SP_Percent := PID_PV_UlazTanka.Out;
			_02_PG_PV02:
				PGRad_Cmd.PropVentili.PV02.SP_Percent := PID_PV_UlazTanka.Out;
		END_CASE
	END_IF

	(* -------------------------------------------------------------------------- *)
	(* 7) Adapter RETAIN ulaznih ventila                                         *)
	(* -------------------------------------------------------------------------- *)
	(* Medjusobno iskljucenje V01/V02 stiti od paralelnog spajanja dva izvora. *)
	IF PGRad.CmdRetain.V01_Open AND PGRad.CmdRetain.V02_Open THEN
		PGRad.CmdRetain.V01_Open := FALSE;
		PGRad.CmdRetain.V02_Open := FALSE;
		FaultLatched := TRUE;
		FaultCode := 10;
		FaultText := 'PG_V01 i PG_V02 istovremeno zahtevani';
	END_IF;

	(* -------------------------------------------------------------------------- *)
	(* 8) Procesni status za Communication/HMI task                              *)
	(* -------------------------------------------------------------------------- *)
	(* Enum State se preslikava u stabilan brojcani status AsIMA/HMI ugovora. *)
	CASE State OF
		PG_01_Priprema_BRB2:
			PGRad_Status.State := 1;
			PGRad_Status.StateComment := 'STANJE: PRIPREMA BRB2';
		PG_02_Rad_BRB2:
			PGRad_Status.State := 2;
			PGRad_Status.StateComment := 'STANJE: RAD BRB2';
		PG_03_Zaustavljanje_BRB2:
			PGRad_Status.State := 3;
			PGRad_Status.StateComment := 'STANJE: ZAUSTAVLJANJE BRB2';
		PG_11_Priprema_IEBKB1:
			PGRad_Status.State := 11;
			PGRad_Status.StateComment := 'STANJE: PRIPREMA IEBKB1';
		PG_12_Rad_IEBKB1:
			PGRad_Status.State := 12;
			PGRad_Status.StateComment := 'STANJE: RAD IEBKB1';
		PG_13_Zaustavljanje_IEBKB1:
			PGRad_Status.State := 13;
			PGRad_Status.StateComment := 'STANJE: ZAUSTAVLJANJE IEBKB1';
	ELSE
		PGRad_Status.State := 0;
		PGRad_Status.StateComment := 'STANJE: STANDBY';
	END_CASE
	PGRad_Status.Substep := Substep;

	CASE State OF
		PG_00_Stand_By:
			PGRad_Status.SubstepComment := 'PODKORAK: Ceka komandu START';

		PG_01_Priprema_BRB2:
			CASE Substep OF
				0: PGRad_Status.SubstepComment := 'PODKORAK: Ulazak u pripremu BRB2';
				1: PGRad_Status.SubstepComment := 'PODKORAK: Ceka zatvaranje PG_V01';
				2: PGRad_Status.SubstepComment := 'PODKORAK: Ceka otvaranje PG_V02';
				3: PGRad_Status.SubstepComment := 'PODKORAK: Ispiranje BRB2 grane';
				4: PGRad_Status.SubstepComment := 'PODKORAK: Priprema ulaza prihvatnog tanka';
				5: PGRad_Status.SubstepComment := 'PODKORAK: Mek prelaz pritiska PG_PV05';
				6: PGRad_Status.SubstepComment := 'PODKORAK: Punjenje prihvatnog tanka';
			ELSE
				PGRad_Status.SubstepComment := 'PODKORAK: Nepoznata priprema BRB2';
			END_CASE

		PG_02_Rad_BRB2:
			IF Substep = 0 THEN
				PGRad_Status.SubstepComment := 'PODKORAK: Pokretanje izlazne pumpe';
			ELSE
				PGRad_Status.SubstepComment := 'PODKORAK: Regulacija i odrzavanje rada';
			END_IF

		PG_03_Zaustavljanje_BRB2:
			PGRad_Status.SubstepComment := 'PODKORAK: Kontrolisano zaustavljanje BRB2';

		PG_11_Priprema_IEBKB1:
			CASE Substep OF
				0: PGRad_Status.SubstepComment := 'PODKORAK: Ulazak u pripremu IEBKB1';
				1: PGRad_Status.SubstepComment := 'PODKORAK: Ceka zatvaranje PG_V02';
				2: PGRad_Status.SubstepComment := 'PODKORAK: Ceka otvaranje PG_V01';
				3: PGRad_Status.SubstepComment := 'PODKORAK: Ceka pocetak dotoka IEBKB1';
				4: PGRad_Status.SubstepComment := 'PODKORAK: Punjenje prihvatnog tanka';
			ELSE
				PGRad_Status.SubstepComment := 'PODKORAK: Nepoznata priprema IEBKB1';
			END_CASE

		PG_12_Rad_IEBKB1:
			IF Substep = 0 THEN
				PGRad_Status.SubstepComment := 'PODKORAK: Pokretanje izlazne pumpe';
			ELSE
				PGRad_Status.SubstepComment := 'PODKORAK: Regulacija i odrzavanje rada';
			END_IF

		PG_13_Zaustavljanje_IEBKB1:
			CASE Substep OF
				0: PGRad_Status.SubstepComment := 'PODKORAK: Ulazak u zaustavljanje IEBKB1';
				1: PGRad_Status.SubstepComment := 'PODKORAK: Ceka prestanak dotoka IEBKB1';
				2: PGRad_Status.SubstepComment := 'PODKORAK: Ceka zatvaranje PG_V05';
				3: PGRad_Status.SubstepComment := 'PODKORAK: Ceka zatvaranje PG_V01';
			ELSE
				PGRad_Status.SubstepComment := 'PODKORAK: Nepoznat stop IEBKB1';
			END_CASE

	ELSE
		PGRad_Status.SubstepComment := 'PODKORAK: Nepoznato stanje sistema';
	END_CASE
	PGRad_Status.Fault := FaultLatched;
	PGRad_Status.FaultCode := FaultCode;

END_PROGRAM
```

#### FLOW_CHART_MASTER.md
~~~~markdown
# Podstanica grejanja Kotlarnica Banja — dijagram rada sistema

> **Verzija:** 0.9 (draft za pregled i overu) • **Datum:** 2026-09-02 • **Autor:** Predrag • **Status:** draft za investitorsku i tehničku overu

> Dokument opisuje **kako rade dva PLC-a** koja zajedno kontrolišu podstanicu:
> - **PLC 1 — PT_KB_V01** kontroliše samu podstanicu (`PG_KB`).
> - **PLC 2 — BRB2_1** kontroliše bunar (`BRB2_rad`).
>
> Dva PLC-a razmenjuju podatke preko optičke veze (protokol AsIMA).

---

## Rečnik pojmova

| Pojam | Značenje |
|---|---|
| **BRB2** | Termalni izvor 2 — kompletan sistem: bunar sa vlastitim pumpama i **sopstvenim PLC-om (`BRB2_1`)**. Komunicira sa podstanicom preko AsIMA. |
| **IEBKB1** | Termalni izvor — takođe kompletan sistem: bunar sa vlastitim pumpama i **sopstvenim PLC-om**. Komunikacija sa podstanicom preko AsIMA (planirano). |
| **PLC 1 / PLC 2** | PLC 1 = kontroler podstanice (`PT_KB_V01`, projekat `PG_KB`). PLC 2 = kontroler bunara BRB2 (`BRB2_1`, projekat `BRB2_rad`). |
| **HMI** | Human-Machine Interface — operaterski panel (touch-screen) za komandovanje, prikaz stanja, alarme i unos SP-ova. Svaki PLC ima svoj HMI. |
| **SCADA** | Centralni sistem nadzora — prima podatke sa svih PLC-ova, log, alarmi, trendovi. |
| **PFD / P&ID** | PFD = Process Flow Diagram (konceptualna šema procesa, ovaj dokument). P&ID = Piping and Instrumentation Diagram (detaljna inženjerska šema — zaseban dokument). |
| **PV (Process Variable)** | **Merena** vrednost koju regulator poredi sa SP-om (npr. PV = trenutni nivo tanka, SP = zadati nivo tanka). |
| **ISA S5.1 prefiksi** | `TT` = temperatura, `PT` = pritisak, `FT`/`MP` = protok, `LS` = nivo (switch, digitalni), `PTNS` = pritisak niskog opsega. |
| **Interlock** | Logički uslov koji **mora biti ispunjen** pre nego što se određena akcija dozvoli (otvaranje ventila, start pumpe, prelaz u sledeći korak). Ako uslov nije ispunjen — akcija se blokira i sistem čeka ili odlazi u kontrolisano zaustavljanje. **Primer:** `PG_V01` sme da se otvori **samo ako je `PG_V02` zatvoren** — nikad oba istovremeno (razdvaja sistem pod nadpritiskom BRB2 od sistema bez nadpritiska IEBKB1, sprečava curenje i mešanje). |
| **SP (SetPoint)** | Zadata vrednost regulacije (npr. `SetPritisakPotisa = 5.5 bar`). Regulator održava mernu vrednost oko SP-a. |
| **RETAIN** | Promenljiva koja se **čuva u PLC memoriji i posle nestanka struje** — kad se PLC ponovo pokrene, vrednost je ista kao pre nestanka. Koristi se za selektore operatera (izvor, mod pumpe...) i za brojače faultova. |
| **AsIMA** | Protokol razmene podataka između dva B&R PLC-a preko optičke veze. U ovom projektu — između podstanice (`PT_KB_V01`) i bunara (`BRB2_1`). |
| **Fault (softverski / hitni)** | Softverski = otklonjivo, sistem pokušava retry 3× pa ide u zaustavljanje. Hitni = trenutno gašenje bez retry-a (npr. prepun tank, pritisak preko limita, kritični senzor izgubljen). Reset se daje sa HMI. |
| **Kontrolisano zaustavljanje** | Uređena sekvenca gašenja: rampa pumpi naniže, sekvencijalno zatvaranje ventila, drenaža po potrebi, prelaz u `Stand_By`. **Suprotno HITNOM gašenju** koje je trenutni stop svih aktuatora. |

---

## A. Šema procesa (konceptualni PFD)

> **KRITIČNI INTERLOCK:** `PG_V01` (IEBKB1 ulaz) i `PG_V02` (BRB2 ulaz) **nikad ne smeju biti istovremeno otvoreni**. Uslov za otvaranje bilo kog od njih je da je onaj drugi **zatvoren**. Razlog: razdvaja se sistem pod nadpritiskom (BRB2) od sistema bez nadpritiska (IEBKB1) — sprečava curenje i mešanje.

```
                    ┌── PG_PV05 ──> DRENAŽNI KANAL
                    │      • ispiranje: čeka T na TT_PG_07 ≥ 60 °C (SP sa HMI)
                    │      • drži pritisak dolaza BRB2 ≥ 5 bar (kad su ventili tanka zatvoreni)
                    │      • drži do 6.5 bar (kad su ventili tanka aktivni — štiti izmenjivače)
                    │      • anti-hidraulički udar: PT_PG_06 > 6.5 bar → auto open
                    │
BRB2 ulaz ──────────┤
(optika + komunikacija ka BRB2 PLC)
                    │                          ┌─ PG_V06 ─ PG_PV01 ─┐
                    └── PG_V02 ────────────────┤                    ├──┐
                                               └─ PG_V07 ─ PG_PV02 ─┘  │
                                                                       ├──> Prihvatni tank
IEBKB1 ulaz ──> PG_V01 ──> PG_V05 ─────────────────────────────────────┘
(optika + komunikacija ka IEBKB1 PLC)  (BYPASS ON/OFF, samo u IEBKB1 modu — direktno u tank, zaobilazi PG_PV01/PV02)
```

> **Važno o ulaznim ventilima:** `PG_V01` i `PG_V02` su **elektromotorni leptir ventili DN150** (`2×DO + 4×DI` po ventilu). Za razliku od pneumatskih (koji su „trenutni"), ovi imaju **hod 15–25 s** od komande do krajnjeg položaja. Interlock i timeout-e u E tabeli su podešeni prema tome. Svi ostali automatski ventili u sistemu (`PG_V03/V04/V05/V06/V07`, `PG_PV05`) su pneumatski (brz odziv < 1 s).

**Senzori na tanku** (nisu u state mašini — merenje/signalizacija):

- `LS_PG_01` — level switch, hi/lo signalizacija
- `TT_PG_03` — temperatura na dnu tanka
- `PTNS_PG_01` — pritisak na dnu tanka
- `PTNS_PG_02` — pritisak vrha tanka (vazdušni prostor)
- `NivoTanka = f(PTNS_PG_01 − PTNS_PG_02)` — izračunata vrednost, koristi se kao PV za regulaciju nivoa

**Izlazna sekcija (od tanka ka potrošačima):**

```
                     ┌── Pu_PG_01 ── PG_V03 ──┐
tank izlaz ─────────┤                          ├──> potis (PT_PG_05, MP_PG_01) ──> ka potrošačima
                     └── Pu_PG_02 ── PG_V04 ──┘  (SP prema `RegulacionaVarijanta` — vidi F.1)
```

Redosled: `tank izlaz` → račva → `Pu_PG_01/02` → `PG_V03/V04` → spajanje → `PT_PG_05`, `MP_PG_01` → potrošači.

### Ključni senzori

> **Napomena:** opsezi su preuzeti iz P&ID export-a *Podstanica 2026-09-01* (spisak uređaja i mernih instrumenata). Softver čita 16-bit skalirane vrednosti prema definiciji u `Types.typ`.

| Oznaka | Značenje | Opseg / jed. |
|---|---|---|
| `TT_PG_07` | Temperatura na drenaži iza `PG_PV05` — uslov za završetak ispiranja (SP = 60 °C, podesivo sa HMI). *Naziv rezervisan; senzor još nije ucrtan na aktuelnom P&ID-u; tip: Easytemp TMR35.* | 0–120 °C |
| `T_Sek_Izl` (generički) | Temperatura sekundara na izlazu iz velikog izmenjivača — PV za mod `temperatura`. **Izvor još nije fiksiran** (opcije: direktno merenje ili preko komunikacije). | TBD °C |
| `PT_PG_06` | Pritisak dolazne magistrale (pre `PG_V02`, na BRB2 ulazu) — anti-hidraulički udar i praćenje ulaznog pritiska. Tip: Cerabar PMP23. | −1–9 bar |
| `PT_PG_05` | Pritisak potisa iza pumpi `Pu_PG_01/02` — SP = `SetPritisakPotisa` (1–1.5 bar u modu `pritisak`). Tip: Cerabar PMP23. | −1–9 bar |
| `MP_PG_01` | Elektromagnetni merač protoka na potisu (donja/gornja granica u modu `pritisak`, monitoring uvek). Tip: Promag H10 DN065. | 0–72 m³/h (0–20 l/s) |
| `PTNS_PG_01` | Pritisak na **dnu** prihvatnog tanka (hidrostatički stub + P vazdušnog prostora). Tip: Cerabar niskog opsega. | −100…300 mbar |
| `PTNS_PG_02` | Pritisak u **vazdušnom prostoru** na vrhu prihvatnog tanka. **Nije potvrđen u trenutnom P&ID export-u — verifikovati sa projektantom.** | −100…300 mbar (očekivano) |
| `NivoTanka` (izračunata) | Nivo vode u prihvatnom tanku = f(`PTNS_PG_01` − `PTNS_PG_02`), preveden u metre. **Logička promenljiva za regulaciju** (ciljno 1.5 m, min 0.9 m, max 2.5 m). | 0–3 m |
| `LS_PG_01` | **Level switch** — diskretni prekidač za signalizaciju prepunjenja / niskog nivoa. **NE koristi se za regulaciju**, samo kao HW zaštita. Tip: Liquipoint FTW23. | digital |

### Izlazne pumpe podstanice (parametri iz P&ID)

- **`Pu_PG_01`, `Pu_PG_02`** — Grundfoss CR45-2A-F-A-E-H00E, vertikalne višestepene centrifugalne.
- **Radni opseg protoka: `MinFR_Pumpe` = 2 l/s, `MaxFR_Pumpe` = 16.2 l/s** (koristi se kao clamp u F.1).
- Signali: `1 x AO 4–20 mA` (zadata frekvencija / brzina), `1 x DI` (radi/stoji), `2 x DO` (start, reset).

### Ostali uređaji na razmenjivačima (van PG_KB regulacije)

Na P&ID-u postoje još senzori i aktuatori na strani razmenjivača koji **nisu deo state-mašine `PG_KB`** — koriste ih zasebni regulacioni krugovi (grejanje objekata, odzraka, higijena). Popisani su ovde samo radi jasnoće da se ne pomešaju sa signalima iz D.1 tabele:

| Oznaka | Namena |
|---|---|
| `TT_PG_05` | Temperatura na razmenjivačima (kandidat za `T_Sek_Izl` — vidi napomenu iznad). |
| `PT_PG_01/02/03` | Pritisci na razmenjivačima (monitoring, ne uđu u D.1). |
| `LS_PG_02/03` | Level switch na razmenjivačima. |
| `PG_PV03`, `PG_PV04` | Membranski proporcionalni ventili Burkert DN025 (odzraka i regulacija razmenjivača). |

### Selektori operatera (RETAIN — čuvaju se posle nestanka struje)

| Selektor | Vrednosti | Napomena |
|---|---|---|
| Izvor termalne vode | `nijedan` · `BRB2` · `IEBKB1` | Vidi F.2. |
| Regulaciona varijanta | `neaktivan` · `pritisak` · `protok` · `temperatura` | Vidi F.1. `temperatura` uslovna (izvor `T_Sek_Izl` TBD). |
| Aktivna izlazna pumpa | `Pu_PG_01` · `Pu_PG_02` | 1 radi, 1 rezerva; auto rotacija po satima rada. |
| Aktivni prop. ventil ulaza tanka | `PG_PV01` · `PG_PV02` | 1 aktivan, 1 rezerva; auto rotacija po satima rada. |
| AutoRestart posle nestanka struje | `OFF` · `ON` | ON → odloženi start 60 s pa auto `KomandaStart`. |

---

## B. PLC 1 — Podstanica (`PT_KB_V01 / PG_KB`)

```mermaid
stateDiagram-v2
    direction TB
    [*] --> PG_00_Stand_By

    PG_00_Stand_By --> PG_01_Priprema_BRB2 : izabran BRB2 + Start
    PG_00_Stand_By --> PG_11_Priprema_IEBKB1 : izabran IEBKB1 + Start

    PG_01_Priprema_BRB2 --> PG_02_Rad_BRB2 : sistem spreman
    PG_01_Priprema_BRB2 --> PG_03_Zaustavljanje_BRB2 : Stop / Fault

    PG_02_Rad_BRB2 --> PG_03_Zaustavljanje_BRB2 : Stop / Fault / promena izvora

    PG_03_Zaustavljanje_BRB2 --> PG_00_Stand_By : zaustavljanje završeno

    PG_11_Priprema_IEBKB1 --> PG_12_Rad_IEBKB1 : sistem spreman
    PG_11_Priprema_IEBKB1 --> PG_13_Zaustavljanje_IEBKB1 : Stop / Fault

    PG_12_Rad_IEBKB1 --> PG_13_Zaustavljanje_IEBKB1 : Stop / Fault / promena izvora
    PG_12_Rad_IEBKB1 --> PG_14_Transfer_IEBKB1_BRB2 : BRB2 spreman + IEB interfejs OK + komanda transfer

    PG_14_Transfer_IEBKB1_BRB2 --> PG_02_Rad_BRB2 : transfer zavrsen
    PG_14_Transfer_IEBKB1_BRB2 --> PG_13_Zaustavljanje_IEBKB1 : IEB stop / V05 / V01 greska
    PG_14_Transfer_IEBKB1_BRB2 --> PG_03_Zaustavljanje_BRB2 : V02 / BRB2 protok greska

    PG_13_Zaustavljanje_IEBKB1 --> PG_00_Stand_By : zaustavljanje završeno
```

### B.1 Šta radi svaki korak

| Korak | Opis |
|---|---|
| `PG_00_Stand_By` | Mirovanje. Sve pumpe stoje; ventili tanka (`PG_V06/V07`, `PG_PV01/02`), izlazni (`PG_V03/V04`) i bypass (`PG_V05`) su zatvoreni. **Ulazni ventili `PG_V01` i `PG_V02` prate `SelektovaniIzvor` (RETAIN):** ako je izabran BRB2 → `PG_V02` otvoren i `PG_V01` zatvoren; ako je izabran IEBKB1 → `PG_V01` otvoren i `PG_V02` zatvoren; ako izvor nije izabran → oba zatvorena. Interlock (nikad oba istovremeno otvorena) uvek važi. Sistem čeka komandu Start sa HMI. |
| `PG_01_Priprema_BRB2` | **Prvi uslov (interlock):** proverava da je `PG_V01` = zatvoren (razdvajanje sistema pod nadpritiskom od sistema bez nadpritiska). Ako nije — blok, greška, ne otvara ništa. Zatim **osigurava da je `PG_V02` otvoren** (obično već jeste iz Stand_By-a jer je BRB2 izabran); pušta bunar preko `PG_PV05` na drenažu, čeka da `TT_PG_07` dostigne 60 °C. Zatim preusmerava na tank (otvara `PG_V06/07` i aktivni `PG_PV01/02`), pali izabranu izlaznu pumpu `Pu_PG_01/02`. **Kad pumpa ustali regulaciju na svom SP-u prema aktivnoj `RegulacionaVarijanta` (F.1) — sistem ulazi u radno stanje.** |
| `PG_02_Rad_BRB2` | Rad sa BRB2 kao izvorom. **`PG_PV01/PV02` NE regulisu protok** — samo održavaju bezbedan pritisak u cevovodu (štite izmenjivače i tank). Ko šta drži zavisi od `RegulacionaVarijanta` (F.1): u `pritisak` varijanti BRB2 drži `NivoTanka` a pumpe drže `PT_PG_05`; u `protok` BRB2 drži svoj FT a pumpe drže `NivoTanka`; u `temperatura` BRB2 juri `T_Sek_Izl` a pumpe kombinovano drže nivo i pritisak potisa (radi zaštite od prelivanja tanka). Anti-udar: `PG_PV05` otvara auto kad `PT_PG_06` > 6.5 bar. |
| `PG_03_Zaustavljanje_BRB2` | Smanjuje protok, zatvara tank granu, gasi izlaznu pumpu, po potrebi zatvara `PG_V02` (samo ako se izvor menja u `Stand_By`-u). Šalje BRB2 komandu za gašenje bunara. Kad je gotovo — sistem se vraća u `PG_00_Stand_By`. |
| `PG_11_Priprema_IEBKB1` | **Prvi uslov (interlock):** proverava da je `PG_V02` = zatvoren (razdvajanje sistema pod nadpritiskom od sistema bez nadpritiska). Ako nije — blok, greška, ne otvara ništa. Zatim **osigurava da je `PG_V01` otvoren** (obično već jeste iz Stand_By-a jer je IEBKB1 izabran) i otvara bypass `PG_V05` ka tanku, pušta IEBKB1 pumpu, čeka punjenje tanka do 1.0 m. Startuje izlaznu pumpu. **Kad pumpa ustali regulaciju na svom SP-u prema aktivnoj `RegulacionaVarijanta` (F.1) — sistem ulazi u radno stanje.** |
| `PG_12_Rad_IEBKB1` | Rad sa IEBKB1 kao izvorom. `PG_V01` je otvoren i IEBKB1 nastavlja punjenje tanka preko `PG_V05`. Komanda `KomandaPripremaBRB2` nezavisno pokreće BRB2 prema drenaži dok `PG_V02` ostaje zatvoren. Priprema potvrđuje pumpu, protok, minimalno trajanje i `TT_PG_07`; `KomandaNastavak` može preskočiti samo temperaturni uslov, ne i potvrdu protoka. |
| `PG_14_Transfer_IEBKB1_BRB2` | Guarded transfer bez prekida rada izlazne pumpe: opoziva zahtev IEBKB1 i čeka nulti protok, zatvara `PG_V05`, zatvara i potvrđuje `PG_V01`, pa tek zatim otvara `PG_V02`. U završnom podkoraku istovremeno radi rampa `PG_PV05/PT06` i regulacija aktivnog `PG_PV01/PV02` prema `PT04`; po potvrđenom BRB2 protoku i zatvorenom `PG_PV05` prelazi u `PG_02_Rad_BRB2`. |
| `PG_13_Zaustavljanje_IEBKB1` | Smanjuje protok IEBKB1, zatvara bypass `PG_V05`, gasi izlaznu pumpu, po potrebi zatvara `PG_V01` (samo ako se izvor menja u `Stand_By`-u). Kad je gotovo — sistem se vraća u `PG_00_Stand_By`. |

> **Važno o prelazu između izvora:** direktan IEBKB1 → BRB2 transfer dozvoljen je samo kada su `BRB2Ready`, `InterfaceReady`, `CommValid` i `HeartbeatValid` potvrđeni i nema udaljenog fault-a. Bez kompletnog budućeg IEBKB1 statusnog ugovora komanda transfera ostaje blokirana. IEBKB1 PLC se ovom implementacijom ne menja.

**Auto-restart posle nestanka struje:** sistem uvek startuje iz `PG_00_Stand_By`. Ponašanje kontroliše HMI selektor `AutoRestart` (RETAIN):
- **`AutoRestart = OFF`** — sistem ostaje u `Stand_By`, čeka manuelnu komandu Start sa HMI-ja.
- **`AutoRestart = ON`** — po isteku **odloženog starta 60 s** sistem automatski šalje `KomandaStart` prema poslednjem RETAIN izboru (`SelektovaniIzvor`, `RegulacionaVarijanta`) i prolazi kroz normalnu Pripremu → Rad. Odloženi start se prekida ako se u tih 60 s pojavi Fault ili operater lokalno pritisne Stop.

---

## C. PLC 2 — Bunar BRB2 (`BRB2_1 / BRB2_rad`)

```mermaid
stateDiagram-v2
    direction TB
    [*] --> B00_StandBy

    B00_StandBy --> B10_Priprema_Hotel : Start + odredište Hotel/PG
    B00_StandBy --> B15_Priprema_IEBKB1 : Start + odredište IEBKB1

    B10_Priprema_Hotel --> B20_Rad_Hotel : sistem spreman
    B10_Priprema_Hotel --> B30_Zaustavljanje_Hotel : Stop / Fault

    B15_Priprema_IEBKB1 --> B25_Rad_IEBKB1 : sistem spreman
    B15_Priprema_IEBKB1 --> B35_Zaustavljanje_IEBKB1 : Stop / Fault

    B20_Rad_Hotel --> B30_Zaustavljanje_Hotel : Stop / Fault
    B25_Rad_IEBKB1 --> B35_Zaustavljanje_IEBKB1 : Stop / Fault

    B30_Zaustavljanje_Hotel --> B00_StandBy : zaustavljanje završeno
    B35_Zaustavljanje_IEBKB1 --> B00_StandBy : zaustavljanje završeno
```

### C.1 Šta radi svaki korak

| Korak | Opis |
|---|---|
| `B00_StandBy` | Mirovanje. Bunar ne radi, oba izlazna ventila zatvorena: `RB2_V01` (izlaz ka IEBKB1 grani) i `RB2_V02` (izlaz ka podstanici PG_KB). Sistem čeka izbor odredišta i komandu Start (od PG_KB preko IMA ili lokalno). |
| `B10_Priprema_Hotel` | Priprema za slanje vode ka podstanici. Verifikuje interlockove, startuje pumpu bunara na 20 Hz (rampa 0.5 Hz/s do izjednačavanja pritisaka), otvara **`RB2_V02`** (ventil ka podstanici PG_KB), prati pritisak **`Pt_RB2_2`** dok ne dostigne 5 bar. |
| `B15_Priprema_IEBKB1` | Priprema za slanje vode ka IEBKB1. Verifikuje interlockove, otvara **`RB2_V01`** (jedini izlaz ka IEBKB1 grani), startuje pumpu bunara. **Nema praćenja pritiska** — cevovod ka IEBKB1 nije opremljen mernom instrumentacijom; spremnost za rad se dobija po komandi/signalu od IEBKB1 kontrolera (ili istekom fiksnog vremena rampe pumpe). |
| `B20_Rad_Hotel` | Rad ka podstanici. Frekvencija pumpe se reguliše prema odabranoj varijanti: **pritisak** (PG diktira), **protok** (BRB2 fiksni 6 l/s) ili **temperatura/snaga**. Dvosmerno mirror-uje stanje sa PG_KB preko IMA. |
| `B25_Rad_IEBKB1` | Rad ka IEBKB1 preko `RB2_V01`. Uvek regulacija po protoku. **Nema praćenja pritiska** na potisnoj strani ka IEBKB1. |
| `B30_Zaustavljanje_Hotel` | Rampa pumpe naniže (0.25 Hz/s), održava pritisak 5.2 bar dok protok ne padne na 0. Zatvara `RB2_V02`, gasi pumpu. Kad je gotovo — sistem se vraća u `B00_StandBy`. |
| `B35_Zaustavljanje_IEBKB1` | Rampa pumpe naniže do 0 (fiksno vreme rampe, bez povratne sprege po pritisku). Zatvara `RB2_V01`, gasi pumpu. Kad je gotovo — sistem se vraća u `B00_StandBy`. |

> **Važno o odabiru odredišta:** odredište (podstanica PG_KB vs IEBKB1) se bira **pre** Pripreme. Priprema ka PG_KB otvara `RB2_V02` i regulisano prati pritisak `Pt_RB2_2` (5 bar). Priprema ka IEBKB1 otvara `RB2_V01` i **radi bez povratne sprege po pritisku** — cevovod ka IEBKB1 nema mernu instrumentaciju. Promena odredišta se dešava **samo iz `B00_StandBy`-a** (nema prečice iz jednog Zaustavljanja u drugu Pripremu). **Nema zajedničke izolacije bunara** — pumpa `Pu_RB2_01/02` je direktno spojena na razvod, tako da su izlazni ventili grana jedini uređaji koji fizički razdvajaju granu.

---

## D. Šta razmenjuju PLC 1 i PLC 2 (AsIMA)

> Filozofija: **sve vrednosti idu na obe strane** (optika je brza i pouzdana, korisno za HMI vizualizaciju na obe lokacije).

### D.1 PG_KB → BRB2 (šta podstanica šalje bunaru)

| Signal | Namena |
|---|---|
| `SelektovaniIzvor`, `RegulacionaVarijanta` | Ogledalo selektora sa HMI podstanice. |
| `KomandaStart`, `KomandaStop` | Komanda bunaru iz PG_KB state mašine. |
| `SpremanZaBRB2` | Podstanica javlja da je spremna da prihvati vodu (nivo, pritisak, nema fault-a). |
| `Sens.*` (`NivoTanka`, `LS_PG_01`, `PT_PG_05`, `MP_PG_01`, `TT_PG_07`, `PT_PG_06`, `PTNS_PG_01`, `PTNS_PG_02`) | Sve merne vrednosti — za HMI na BRB strani. |
| `Act.*` (otvor PG_PV01/02/05, FR izlaznih pumpi) | Trenutno stanje aktuatora — za HMI. |

### D.2 BRB2 → PG_KB (šta bunar šalje podstanici)

| Signal | Namena |
|---|---|
| `PumpaAktivna`, `FR_Actual` | Status bunarske pumpe. |
| `FaultLatched`, `FaultCode` | Ako BRB2 ima grešku — PG ide u kontrolisano zaustavljanje. |
| `Sens.*` (PT bunara, FT bunara, TT bunara) | Merne vrednosti sa bunara — za HMI podstanice. |
| `Act.*` (Pumpa_snaga, otvor RB2_V01/02) | Trenutno stanje aktuatora bunara. |

**Ako AsIMA veza padne > 5 s** → obe strane idu u kontrolisano zaustavljanje.

### D.3 PG_KB → IEBKB1 (planirano — ista logika kao D.1)

Struktura poruke identična kao D.1. Razlika u parametrizaciji: IEBKB1 grana ima ograničen maksimalni protok, pa se `SP_Protok` pre slanja clamp-uje na `MaxProtok_IEBKB1` (RETAIN konstanta iz projekta / HMI).

### D.4 IEBKB1 → PG_KB (planirano — ista logika kao D.2)

Struktura poruke identična kao D.2. Ista fault i timeout logika: **AsIMA link IEBKB1 pao > 5 s** → kontrolisano zaustavljanje na obe strane.

---

## E. Greške i reset

Svaki uslov greške ima definisan SP: prag vrednosti i/ili trajanje (debounce) pre okidanja.

| Greška | Uslov / SP | Reakcija |
|---|---|---|
| Interlock nije OK u Pripremi | invalid interlock signal (nedostatak potvrde `CLOSED` na drugom ventilu) > **2 s** (V01/V02 su elektromotorni) | Prelaz u Zaustavljanje, čeka reset sa HMI. |
| `PG_V01` ili `PG_V02` ne dostiže krajnji položaj | od komande do potvrde LSU (`OPEN` ili `CLOSED`) > **30 s** | Zaustavljanje, greska, potreban reset i inspekcija ventila. |
| **Interlock `PG_V01` + `PG_V02` istovremeno OPEN** | oba povratna kontakta `= OPEN` > **200 ms** | **HITNO** gašenje: oba ventila CLOSED, sve pumpe STOP, `PG_PV05` OPEN, prelaz u `PG_00_Stand_By` sa lokovanom greškom — zahteva reset i inspekciju. |
| BRB2/IEBKB1 ne odgovara na komandu | odziv na `KomandaStart`/`KomandaStop` > **30 s** | Kontrolisano zaustavljanje. |
| Ispiranje predugo | `TT_PG_07 < 60 °C` posle **10 min** od starta ispiranja | Pauza, retry 3×; posle 3. → zaustavljanje. |
| Nivo tanka previsok | `NivoTanka > 2.5 m` **ili** `LS_PG_01_hi` aktivan > **2 s** | **HITNO:** svi ventili zatvoreni, pumpe stop, `PG_PV05` otvoren. |
| Nivo tanka nizak tokom rada | `NivoTanka < 0.3 m` **ili** `LS_PG_01_lo` aktivan > **30 s** | Pauza, retry 3×; posle 3. → zaustavljanje. |
| Pritisak dolaza previsok | `PT_PG_06 > 8 bar` > **1 s** | **HITNO** gašenje. |
| Alarm izlazne pumpe | trip signal `Pu_PG_01/02` **ili** struja > **120 % In** > **5 s** | Zaustavljanje, retry sa rotacijom pumpi ako je moguće. |
| AsIMA link pao | timeout > **5 s** | Kontrolisano zaustavljanje na obe strane. |
| Kritičan senzor izgubljen | vrednost van opsega (`< 0` ili `> nominalni raspon`) > **2 s** | **HITNO** gašenje. |

**Reset:** operater na HMI daje `KomandaReset`; sistem se vraća u `PG_00_Stand_By` ako je uzrok otklonjen.

**Prijava alarma:** svaka greška se javlja istovremeno na **HMI podstanice (PT_KB)**, **HMI BRB2** i **centralnu SCADA**. Kod, vreme i opis se logiraju lokalno u RETAIN buferu (poslednjih 100 događaja) i šalju u SCADA istoriju.

---

## F. Modovi rada

### F.1 Regulaciona varijanta (`RegulacionaVarijanta`)

Selektor sa HMI, RETAIN. Definiše ko šta reguliše u lancu bunar → tank → bazeni. **Bunar uvek ima ograničenja `Min/MaxProtok` i `Min/MaxFR_Pumpe`.**

| Varijanta | Bunar drži | Pumpe podstanice Pu_PG_01/02 drže | Šta PG_KB šalje bunaru |
|---|---|---|---|
| `pritisak` | `NivoTanka` (željeni nivo u prihvatnom tanku) | `PT_PG_05` = **1–1.5 bar** (pritisak potisa ka bazenima) | `SP_NivoTanka` (a) **ili** `SP_Protok = f(NivoTanka)` (b) — izbor sa HMI |
| `protok` | svoj `FT bunara` = `SP_Protok` (direktno sa HMI) | `NivoTanka` (menjaju svoj protok potisa da drže zadati nivo tanka) | `SP_Protok` direktno sa HMI |
| `temperatura` | podiže `SP_Protok` dok `T_Sek_Izl` ne dostigne `SP_T_Sek_Izl` | kombinovano: primarno `NivoTanka` (jer bunar u traženju temperature može stvoriti prevelik protok i preliti tank), sekundarno `PT_PG_05` kad ima rezerve | PG_KB računa `SP_Protok = f(T_Sek_Izl)`, ograničeno `MaxProtok` odnosno `MaxFR_Pumpe` |

> **Važno:** za IEBKB1 kao izvor sve vrednosti `SP_Protok` se dodatno clamp-uju na `MaxProtok_IEBKB1` (grana ima manji kapacitet od BRB2).
>
> **Napomena o modu `temperatura`:** dostupan je samo kad se fiksira izvor senzora `T_Sek_Izl` (direktno merenje ili preko komunikacije). Do tada je varijanta `temperatura` blokirana na HMI-ju — selektor je vidljiv ali sa oznakom *nedostupno*.

### F.2 Izbor izvora (`SelektovaniIzvor`)

| Vrednost | Ulazna grana | Napomena |
|---|---|---|
| `BRB2` | `PG_V02` OPEN, `PG_V01` CLOSED | Standardni režim — pun kapacitet. |
| `IEBKB1` | `PG_V01` OPEN, `PG_V02` CLOSED, opciono `PG_V05` BYPASS | Ograničen maksimalni protok (`MaxProtok_IEBKB1`). |

**Kritični interlock:** `PG_V01` i `PG_V02` nikada istovremeno otvoreni — hardverska i softverska brava; kršenje → HITNO gašenje (vidi sekciju E).

---

## G. Napomene za nastavak rada

- Detaljne substep-ove svake faze (šta u kom trenutku otvara/zatvara), IMA sequence sa vremenskim redosledom, kompletnu tabelu fault kodova (F01…F70) i status implementacije po fajlovima — vidi `TEHNICKI_DODATAK.md` u istom folderu.
- Kod za state mašine: `Cyclic.st` u [Rad_PG_KB/](.) (PT_KB_V01) i `Cyclic.sfc` u `BRB2_1/Logical/Project/BRB2_rad/`.
- Deklaracije tipova i strukture: `Types.typ` u istim folderima.
~~~~

#### Init.st
```iecst
PROGRAM _INIT
	(* ======================================================================== *)
	(* 1) Inicijalizacija izvrsnog konteksta                                     *)
	(* ======================================================================== *)
	State := PG_00_Stand_By;
	Substep := 0;

	KomandaStart := FALSE;
	KomandaStop := FALSE;
	KomandaReset := FALSE;
	CmdSetDefaultParameters := FALSE;
	IF PGRad.Ctrl.SelektovaniIzvor = _02_IEBKB1 THEN
		SelectIEBKB1 := TRUE;
	ELSE
		SelectIEBKB1 := FALSE;
		PGRad.Ctrl.SelektovaniIzvor := _01_BRB2;
	END_IF;

	FaultLatched := FALSE;
	FaultCode := 0;
	FaultText := '';
	T_PG_V01_Close(IN := FALSE, PT := T#0s);
	T_PG_V02_Open(IN := FALSE, PT := T#0s);
	T_PrelazPV05Cuvar(IN := FALSE, PT := T#0s);
	SP_PV05 := 0.0;
	PV05IspiranjeOtvoreno := FALSE;
	IzlaznaPumpaUStopu := FALSE;

	(* ======================================================================== *)
	(* 2) Inicijalizacija PID parametara proporcionalnih ventila                *)
	(* ======================================================================== *)
	(* PV05 cuva pritisak dolaznog voda, a aktivni ulazni PV odrzava PT04. *)
	PID_PV05.MinOut := 0.0;
	PID_PV05.MaxOut := 100.0;
	PID_PV05.PIDParameters.DerivativeTime := 0.0;
	PID_PV05.PIDParameters.FilterTime := 45.0;
	PID_PV05.PIDParameters.Gain := 1.0;
	PID_PV05.PIDParameters.IntegrationTime := 180.0;
	PID_PV05.Invert := TRUE;
	PID_PV05.Update := TRUE;

	PID_PV_UlazTanka.MinOut := 0.0;
	PID_PV_UlazTanka.MaxOut := 100.0;
	PID_PV_UlazTanka.PIDParameters.DerivativeTime := 0.0;
	PID_PV_UlazTanka.PIDParameters.FilterTime := 45.0;
	PID_PV_UlazTanka.PIDParameters.Gain := 1.0;
	PID_PV_UlazTanka.PIDParameters.IntegrationTime := 180.0;
	PID_PV_UlazTanka.Invert := FALSE;
	PID_PV_UlazTanka.Update := TRUE;

	(* ======================================================================== *)
	(* 3) Obnova RETAIN komandi bistabilnih ulaznih ventila                      *)
	(* ======================================================================== *)
	(* RETAIN polozaji se neposredno prenose na bistabilne ulazne ventile. *)
	PG.Act.AV._1.Open := PGRad.CmdRetain.V01_Open; (* PG_V01: dolaz sa IEBKB1. *)
	PG.Act.AV._2.Open := PGRad.CmdRetain.V02_Open; (* PG_V02: dolaz sa BRB2. *)

	(* ======================================================================== *)
	(* 4) Bezbedan reset neretentivnog upravljackog vektora                      *)
	(* ======================================================================== *)
	PGRad_Cmd.Aktivan := FALSE;
	PGRad_Cmd.Ventili._03_Open := FALSE;
	PGRad_Cmd.Ventili._04_Open := FALSE;
	PGRad_Cmd.Ventili._05_Open := FALSE;
	PGRad_Cmd.Ventili._06_Open := FALSE;
	PGRad_Cmd.Ventili._07_Open := FALSE;

	PGRad_Cmd.PropVentili.PV01.Enable := FALSE;
	PGRad_Cmd.PropVentili.PV02.Enable := FALSE;
	PGRad_Cmd.PropVentili.PV05.Enable := FALSE;
	PGRad_Cmd.AirRelease.PV03.Enable := FALSE;
	PGRad_Cmd.AirRelease.PV04.Enable := FALSE;
	PGRad_Cmd.AirRelease.UseIEBKB1Parameters := FALSE;
	PGRad_Cmd.AirRelease.ResetAll := FALSE;

	PGRad_Cmd.Pumpe._01.Run := FALSE;
	PGRad_Cmd.Pumpe._02.Run := FALSE;
	PGRad_Cmd.PID.Enable := FALSE;
	PGRad_Cmd.PID.ActValue := 0.0;
	PGRad_Cmd.PID.SetValue := 0.0;
	PGRad_Cmd.PID.Invert := FALSE;
	PGRad_Cmd.PID.MaxOut := 0.0;
	PGRad_Cmd.PID.EnableTracking := FALSE;
	PGRad_Cmd.PID.TrackingValue := 0.0;
	PGRad_BRB2Cmd.ZahtevZaustavljanja := FALSE;
	PGRad_BRB2Cmd.VentiliPodstaniceZatvoreni := FALSE;

	(* ======================================================================== *)
	(* 5) Cold-boot provera RETAIN parametara                                   *)
	(* ======================================================================== *)
	(* RETAIN parametri se inicijalizuju i na cold boot-u. *)
	IF (PGRad.Par.SetPritisakPotisa <= 0.0)
		OR (PGRad.Par.MaxFR_Pumpe <= 0.0)
		OR (PGRad.Par.SetPointPritisakPV05Ispiranje <= 0.0)
		OR (PGRad.Par.SetPointPritisakUlazTanka <= 0.0)
		OR (PGRad.Par.TimeSP.PrelazPV05Cuvar_s <= 0.0)
		OR (PGRad.Par.PocetnaFrekvencaIzlaznePumpe <= 0.0)
		OR (PGRad.Par.MaxOtvorPropZaZatvaranje <= 0.0)
		OR (PGRad.Par.TimeSP.OverlapPumpi_s <= 0.0)
		OR (PGRad.Par.TimeSP.AutoRestartDelay_s <= 0.0)
		OR (PGRad.Par.TimeSP.ValvePositionTimeout_s <= 0.0)
		OR (PGRad.Par.TimeSP.InterlockDebounce_s <= 0.0)
		OR (PGRad.Par.AirRelease.BRB2.PV03.NumberOfLS = 0)
		OR (PGRad.Par.AirRelease.BRB2.PV04.NumberOfLS = 0)
		OR (PGRad.Par.AirRelease.IEBKB1.PV03.NumberOfLS = 0)
		OR (PGRad.Par.AirRelease.IEBKB1.PV04.NumberOfLS = 0) THEN
		CmdSetDefaultParameters := TRUE;
	END_IF

END_PROGRAM
```
